ABB RobotStudio station: Cell5678 2025_5_GPA546_A0610_RW7.5.rspag

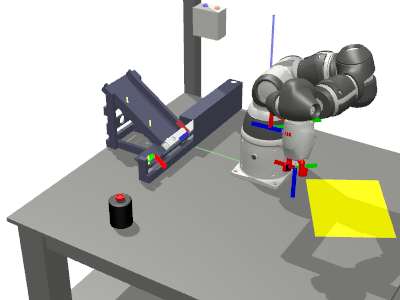
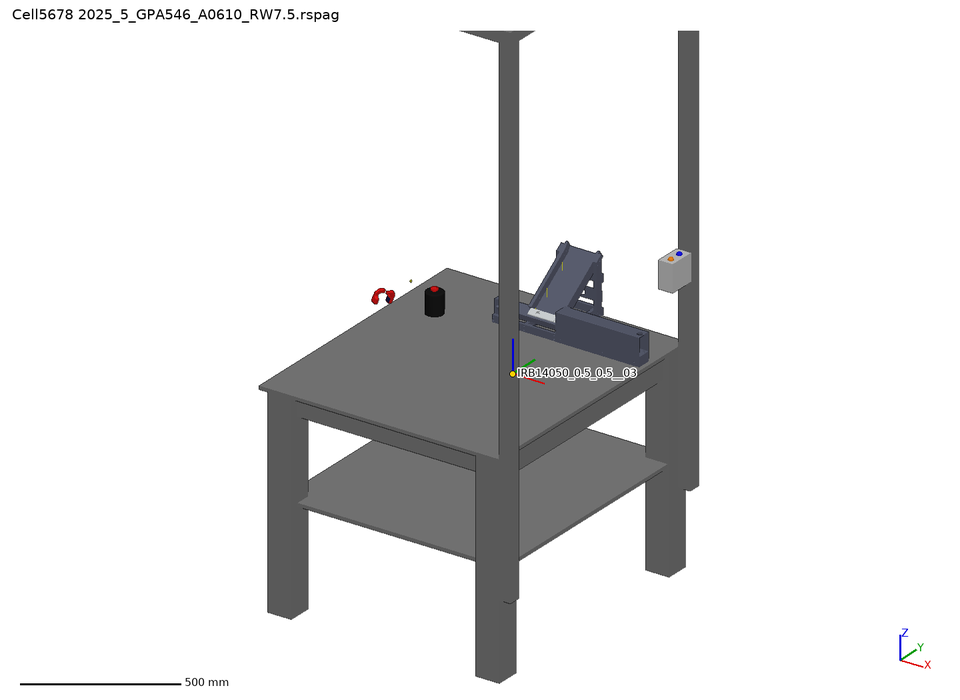
[picture v1: parts stored in the station drawn from their meshes, with robot base, taught points and paths (robot models come from the ABB library and are not in the file)]
--- station ---
Station Cell5678 011021_GPA546_A0610_publ5_1 (saved by RobotStudio 24.2.10821.1)
Controller IRB14050
  mechanical unit ROB_1: IRB14050_0.5_0.5__03, 6 joints, base frame (0, 0, 0) mm
  mechanical unit ROB_1_7: IRB14050_0.5_0.5__03, 1 joints, base frame (0, 0, 0) mm
Layout (positions relative to the parent item):
  - IRB14050_0.5_0.5__03 [mechanism, from %ABB.RobotStudio.Models.IRB14050%\IRB14050_0.5_0.5__03.rslib] at (0, 0, 0) mm; joint values [1.5708, -1.309, 1.5708, 0.3491, -1.5708, -1.2217, 1.5708] (rad or m)
  - Table 1020X900 [part] at (311.38, -523.15, 0.9) mm, rotated rx 0 ry 0 rz 90 deg, size 1020 x 954.9 x 2265 mm
  - Boite Lumière [part] at (359.1, 353.08, 238.5) mm, rotated rx 0 ry 0 rz 90 deg, size 100 x 55 x 100 mm
  - Glissoire_4 [part] at (-154.02, 493.45, 6.79) mm, rotated rx 0 ry 0 rz -90 deg, size 257.5 x 560.4 x 225.6 mm
  - Piston [mechanism, from Libraries\Piston.rslib] at (-154.02, 493.45, 6.79) mm, rotated rx 0 ry 0 rz -90 deg; joint values [0] (rad or m)
  - SC_Gestion_Lampes [smart component]
      signals: DI BlueLampOn, DI YellowLampOn
      connections:
        SC_Gestion_Lampes.BlueLampOn -> Highlighter.Active
        SC_Gestion_Lampes.YellowLampOn -> Highlighter_2.Active
    - Highlighter [smart component, from Components\Highlighter.rslib]
        properties: Object=Lumière Bleu; Color=[0 0 255]; Opacity=255
    - Highlighter_2 [smart component, from Components\Highlighter.rslib]
        properties: Object=Lumière Jaune; Color=[255 50 0]; Opacity=255
  - Lumière Bleu [part] at (10.6, -21.42, 0) mm, rotated rx 0 ry 0 rz -90 deg, size 19.9 x 19.9 x 20 mm
  - Lumière Jaune [part] at (10.6, -21.42, 0) mm, rotated rx 0 ry 0 rz -90 deg, size 19.9 x 19.9 x 20 mm
  - SC_Gestion poussoir [smart component] at (-154.05, 492.67, 6.82) mm, rotated rx 0 ry 0 rz -90 deg
      properties: PartAtPickPoint=(none)
      signals: DI ValveON, DO AtExtend, DO AtRetract, AO BlocAtLow, DO BlocAtHigh, DO NoHoleDetect, DO BlocZS0101, DI Orientation
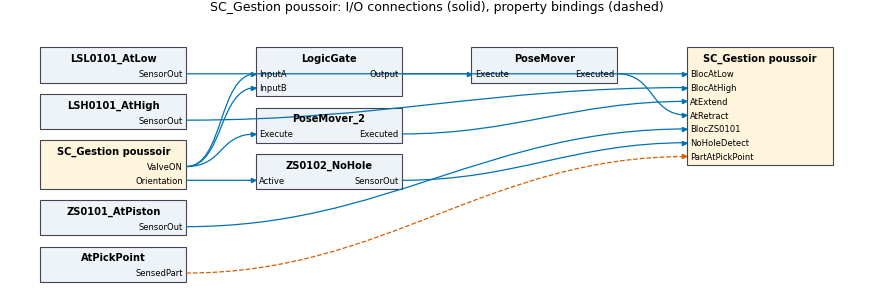
      connections:
        LSL0101_AtLow.SensorOut -> SC_Gestion poussoir.BlocAtLow
        LSH0101_AtHigh.SensorOut -> SC_Gestion poussoir.BlocAtHigh
        LogicGate.Output -> PoseMover.Execute
        SC_Gestion poussoir.ValveON -> LogicGate.InputA
        SC_Gestion poussoir.ValveON -> LogicGate.InputB
        SC_Gestion poussoir.ValveON -> PoseMover_2.Execute
        PoseMover_2.Executed -> SC_Gestion poussoir.AtExtend
        PoseMover.Executed -> SC_Gestion poussoir.AtRetract
        ZS0101_AtPiston.SensorOut -> SC_Gestion poussoir.BlocZS0101
        SC_Gestion poussoir.Orientation -> ZS0102_NoHole.Active
        ZS0102_NoHole.SensorOut -> SC_Gestion poussoir.NoHoleDetect
        AtPickPoint.SensedPart => SC_Gestion poussoir.PartAtPickPoint
    - PoseMover [smart component, from Components\PoseMover.rslib] at (516.34, -722.56, -751.2) mm, rotated rx 0 ry 0 rz -5.2 deg
        properties: Mechanism=Piston; Pose=2; Duration=2
    - PoseMover_2 [smart component, from Components\PoseMover.rslib] at (516.34, -722.56, -751.2) mm, rotated rx 0 ry 0 rz -5.2 deg
        properties: Mechanism=Piston; Pose=3; Duration=2
    - LogicGate [smart component, from Components\LogicGate.rslib] at (516.34, -722.56, -751.2) mm, rotated rx 0 ry 0 rz -5.2 deg
        properties: Operator=NOT; Delay=0
    - ZS0101_AtPiston [smart component, from Components\LineSensor.rslib] at (516.34, -722.56, -751.2) mm, rotated rx 0 ry 0 rz -5.2 deg
        properties: Start=[-0.375541 0.733962 0.796662]; End=[-0.375541 0.733962 0.826662]; Radius=0.001; SensedPart=Bloc_ETS_D0; SensedPoint=[-0.111608673095703 0.283746734619141 0.0522771530151367]; Length=0.03; Tag=(none)
      - _sensorPart_ [part], size 2 x 2 x 30 mm
    - LSL0101_AtLow [smart component, from Components\LineSensor.rslib] at (516.34, -722.56, -751.2) mm, rotated rx 0 ry 0 rz -5.2 deg
        properties: Start=[-0.437628 0.727535 0.840369]; End=[-0.437628 0.727535 0.870369]; Radius=0.001; SensedPart=(none); SensedPoint=[0 0 0]; Length=0.0299999999999999; Tag=(none)
      - _sensorPart_ [part], size 2 x 2 x 30 mm
    - LSH0101_AtHigh [smart component, from Components\LineSensor.rslib] at (516.34, -722.56, -751.2) mm, rotated rx 0 ry 0 rz -5.2 deg
        properties: Start=[-0.520412 0.718966 0.898644]; End=[-0.520412 0.718966 0.928644]; Radius=0.001; SensedPart=(none); SensedPoint=[0 0 0]; Length=0.03; Tag=(none)
      - _sensorPart_ [part], size 2 x 2 x 30 mm
    - ZS0102_NoHole [smart component, from Components\LineSensor.rslib] at (516.34, -722.56, -751.2) mm, rotated rx 0 ry 0 rz -5.2 deg
        properties: Start=[-0.38024951999447 0.783345123820164 0.800380266534001]; End=[-0.367482382887285 0.784507947657669 0.818689278845135]; Radius=0.004; SensedPart=Bloc_ETS_G0; SensedPoint=[-0.0620019989013672 0.283955902099609 0.0559951324462891]; Length=0.0223511046930568; Tag=(none)
      - _sensorPart_ [part], size 19.3 x 9.1 x 22.9 mm
    - AtPickPoint [smart component, from Components\LineSensor.rslib] at (516.34, -722.56, -751.2) mm, rotated rx 0 ry 0 rz -5.2 deg
        properties: Start=[-0.358924 0.623964 0.79302]; End=[-0.358924 0.623964 0.82302]; Radius=0.001; SensedPart=(none); SensedPoint=[0 0 0]; Length=0.03; Tag=(none)
      - _sensorPart_ [part], size 2 x 2 x 30 mm
  - SC_Gestion bloc [smart component]
      signals: DI PistonValve_ON, DI PistonRetracted, DO SimulBlocPoussoir, DI PistonExtended, DI Reinit_Droite, DI Reinit_Gauche, DI Initialisation
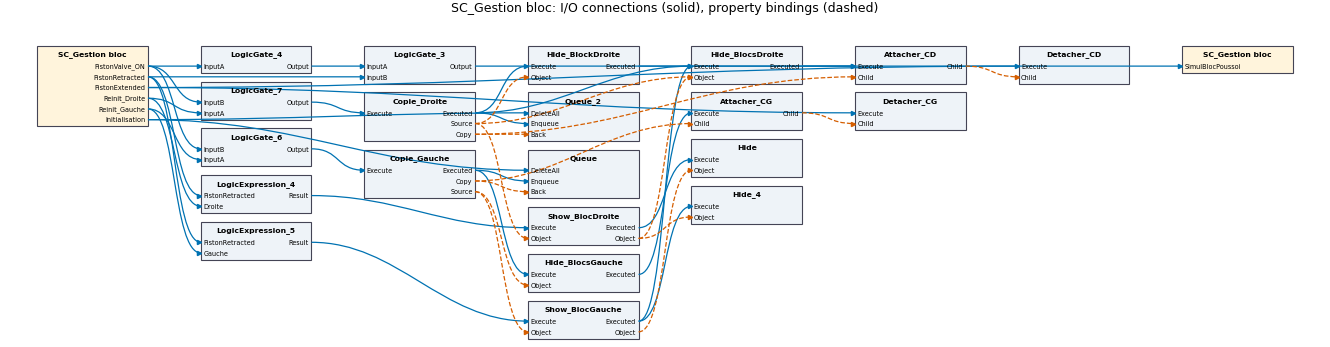
      connections:
        SC_Gestion bloc.PistonValve_ON -> LogicGate_4.InputA
        LogicGate_3.Output -> SC_Gestion bloc.SimulBlocPoussoir
        LogicExpression_4.Result -> Show_BlocDroite.Execute
        LogicExpression_5.Result -> Show_BlocGauche.Execute
        SC_Gestion bloc.PistonRetracted -> LogicExpression_4.PistonRetracted
        SC_Gestion bloc.PistonRetracted -> LogicExpression_5.PistonRetracted
        Copie_Gauche.Executed -> Hide_BlocsGauche.Execute
        SC_Gestion bloc.PistonExtended -> Detacher_CG.Execute
        LogicGate_6.Output -> Copie_Gauche.Execute
        SC_Gestion bloc.PistonValve_ON -> LogicGate_6.InputB
        LogicGate_7.Output -> Copie_Droite.Execute
        SC_Gestion bloc.PistonValve_ON -> LogicGate_7.InputB
        SC_Gestion bloc.PistonExtended -> Detacher_CD.Execute
        SC_Gestion bloc.Reinit_Droite -> LogicExpression_4.Droite
        SC_Gestion bloc.Reinit_Gauche -> LogicExpression_5.Gauche
        LogicGate_4.Output -> LogicGate_3.InputA
        SC_Gestion bloc.PistonRetracted -> LogicGate_3.InputB
        SC_Gestion bloc.Reinit_Gauche -> LogicGate_6.InputA
        SC_Gestion bloc.Reinit_Droite -> LogicGate_7.InputA
        Copie_Droite.Executed -> Hide_BlocsDroite.Execute
        Hide_BlocsDroite.Executed -> Attacher_CD.Execute
        SC_Gestion bloc.Initialisation -> Queue.DeleteAll
        SC_Gestion bloc.Initialisation -> Queue_2.DeleteAll
        Show_BlocDroite.Executed -> Hide.Execute
        Show_BlocGauche.Executed -> Hide_2.Execute
        Hide_BlocsGauche.Executed -> Attacher_CG.Execute
        Copie_Droite.Executed -> Hide_BlockDroite.Execute
        Hide_BlockDroite.Executed -> Attacher_CD.Execute
        Show_BlocGauche.Executed -> Hide_4.Execute
        Copie_Gauche.Executed -> Queue.Enqueue
        Copie_Droite.Executed -> Queue_2.Enqueue
        Attacher_CG.Child => Detacher_CG.Child
        Attacher_CD.Child => Detacher_CD.Child
        Show_BlocGauche.Object => Hide.Object
        Show_BlocDroite.Object => Hide_2.Object
        Copie_Gauche.Copy => Attacher_CG.Child
        Copie_Gauche.Source => Hide_BlocsGauche.Object
        Copie_Gauche.Source => Show_BlocGauche.Object
        Copie_Droite.Source => Show_BlocDroite.Object
        Copie_Droite.Copy => Attacher_CD.Child
        Copie_Droite.Source => Hide_BlocsDroite.Object
        Copie_Droite.Source => Hide_BlockDroite.Object
        Show_BlocDroite.Object => Hide_4.Object
        Copie_Gauche.Copy => Queue.Back
        Copie_Droite.Copy => Queue_2.Back
    - LogicGate_3 [smart component, from Components\LogicGate.rslib]
        properties: Operator=AND; Delay=0
    - LogicGate_4 [smart component, from Components\LogicGate.rslib]
        properties: Operator=NOT; Delay=0
    - Show_BlocDroite [smart component, from Components\Show.rslib]
        properties: Object=Bloc_ETS_D0
    - Show_BlocGauche [smart component, from Components\Show.rslib]
        properties: Object=Bloc_ETS_G0
    - Hide_BlocsGauche [smart component, from Components\Hide.rslib]
        properties: Object=Bloc_ETS_G0
    - LogicExpression_4 [smart component, from Components\LogicExpression.rslib]
        properties: Expression=PistonRetracted and Droite
    - LogicExpression_5 [smart component, from Components\LogicExpression.rslib]
        properties: Expression=PistonRetracted and Gauche
    - Copie_Droite [smart component, from Components\Source.rslib]
        properties: Source=Bloc_ETS_D0; Copy=(none); Parent=(none); Position=[-0.079147 0.2595 0.06725]; Orientation=[0.610865238198015 0 0]; Transient=true; PhysicsBehavior=0
    - Copie_Gauche [smart component, from Components\Source.rslib]
        properties: Source=Bloc_ETS_G0; Copy=(none); Parent=(none); Position=[-0.079147 0.26106 0.06725]; Orientation=[-2.18166156499291 0 3.14159265358979]; Transient=true; PhysicsBehavior=0
    - Attacher_CG [smart component, from Components\Attacher.rslib]
        properties: Parent=L2; Flange=0; Child=(none); Mount=false; Offset=[0 0 0]; Orientation=[0 0 0]
    - Detacher_CG [smart component, from Components\Detacher.rslib]
        properties: Child=(none); KeepPosition=true
    - LogicGate_6 [smart component, from Components\LogicGate.rslib]
        properties: Operator=AND; Delay=0
    - LogicGate_7 [smart component, from Components\LogicGate.rslib]
        properties: Operator=AND; Delay=0
    - Attacher_CD [smart component, from Components\Attacher.rslib]
        properties: Parent=L2; Flange=0; Child=(none); Mount=false; Offset=[0 0 0]; Orientation=[0 0 0]
    - Detacher_CD [smart component, from Components\Detacher.rslib]
        properties: Child=(none); KeepPosition=true
    - Queue [smart component, from Components\Queue.rslib]
        properties: Back=(none); Front=(none); Queue=; NumberOfObjects=0
    - Queue_2 [smart component, from Components\Queue.rslib]
        properties: Back=(none); Front=(none); Queue=; NumberOfObjects=0
    - Hide [smart component, from Components\Hide.rslib]
        properties: Object=Bloc_ETS_G0
    - Hide_BlockDroite [smart component, from Components\Hide.rslib]
        properties: Object=Bloc_ETS_D0
    - Hide_4 [smart component, from Components\Hide.rslib]
        properties: Object=Bloc_ETS_D0
  - Feuille8.5x11 [part, from Libraries\Feuille8.5x11.rslib] at (-117.65, -454.21, 2) mm, rotated rx 0 ry 0 rz 30 deg
  - Smart_Gripper_Group [graphiccomponentgroup] at (-291.1, -222.85, 372.1) mm, rotated rx -165.24 ry 14.08 rz 69.35 deg
    - YuMiFinger_2 [part] at (-0.5, -6.5, 84) mm, rotated rx 0 ry 0 rz 180 deg, size 33.9 x 23.8 x 46.2 mm
    - Smart_Gripper [mechanism] at (0, 0, 0) mm; joint values [0.025] (rad or m)
        TCP Servo at (0, 0, 84) mm
        TCP VaccumOne at (63.5, 18.5, 37.5) mm, rotated rx 0 ry 90 rz 0 deg
        TCP Camera at (-7.3, 28.3, 35.1) mm, rotated rx 0 ry 90 rz 90 deg
        links: HandBase, DownFinger, UpFinger
    - YuMiFinger [part] at (0.5, 6.5, 84) mm, size 33.9 x 23.8 x 46.2 mm
  - CrayonAttache [part] at (-176.86, -64.88, 338.21) mm, rotated rx -31.34 ry -80.07 rz -136.95 deg, size 25 x 25 x 53.7 mm
  - Support_Probe [part] at (-446.5, 212.7, 77.11) mm, size 63.4 x 63.5 x 76.2 mm
  - CrayonDansSupport [part] at (-446.94, 212.7, 84.94) mm, rotated rx 180 ry 0 rz 180 deg, size 25 x 25 x 53.7 mm
  - PadUp [part] at (-346.78, -144.15, -46.95) mm, rotated rx 5.22 ry 23.93 rz 58.66 deg, size 8.7 x 19.9 x 17.8 mm
  - PadDown [part] at (-330.6, -100.22, -58.38) mm, rotated rx 5.22 ry 23.93 rz 58.66 deg, size 8.7 x 19.9 x 17.8 mm
  - Bloc_ETS_G0 [part] at (-79.15, 261.06, 67.25) mm, rotated rx -125 ry 0 rz 180 deg, size 99.6 x 26.5 x 26.5 mm
  - SC_Gestion crayon [smart component]
      signals: DI Succion
      connections:
        ObjectComparer.Output -> LogicGate.InputB
        SC_Gestion crayon.Succion -> LogicGate.InputA
        LogicGate.Output -> Attacher.Execute
        SC_Gestion crayon.Succion -> LogicGate_2.InputA
        LogicGate_2.Output -> Detacher.Execute
        LineSensor.SensedPart => ObjectComparer.ObjectB
        DetecteurCrayon.SensedPart => ObjectComparer_2.ObjectB
        DetecteurCrayon.SensedPart => ObjectComparer_3.ObjectB
        DetecteurCrayon.SensedPart => GetParent.Child
        DetecteurCrayon.SensedPart => ObjectComparer.ObjectB
        ObjectComparer.ObjectA => Attacher.Child
        ObjectComparer.ObjectA => Detacher.Child
    - DetecteurCrayon [smart component, from Components\VolumeSensor.rslib] at (-291.1, -222.85, 372.1) mm, rotated rx -165.24 ry 14.08 rz 69.35 deg
        properties: CornerPoint=[0.0651107378011944 0.0208370386716533 0.0417702285630413]; Orientation=[-1.57722951002103 0.179635421049669 -1.58129130311226]; Length=0.008; Width=0.008; Height=0.001; PartialHit=true; SensedPart=Pneumatic; Tag=(none)
      - _sensorPart_ [part], size 1.1 x 9.3 x 9.3 mm
    - ObjectComparer [smart component, from Components\ObjectComparer.rslib]
        properties: ObjectA=CrayonDansSupport; ObjectB=Pneumatic
    - LogicGate [smart component, from Components\LogicGate.rslib]
        properties: Operator=AND; Delay=0
    - Attacher [smart component, from Components\Attacher.rslib]
        properties: Parent=Pneumatic; Flange=0; Child=CrayonDansSupport; Mount=false; Offset=[0 0 0]; Orientation=[0 0 0]
    - LogicGate_2 [smart component, from Components\LogicGate.rslib]
        properties: Operator=NOT; Delay=0
    - Detacher [smart component, from Components\Detacher.rslib]
        properties: Child=CrayonDansSupport; KeepPosition=true
  - LogicGate [smart component, from Components\LogicGate.rslib]
      properties: Operator=OR; Delay=0
  - Random [smart component, from Components\Random.rslib]
      properties: Value=0.33026239151613; Min=0; Max=1
  - LogicGate_2 [smart component, from Components\LogicGate.rslib]
      properties: Operator=NOT; Delay=0
  - Bloc_ETS_D0 [part] at (-79.15, 281.54, 81.59) mm, rotated rx -55 ry 0 rz 0 deg, size 98 x 25.4 x 25.4 mm
  - ExecuteCommand [smart component, from Components\ExecuteCommand.rslib]
      properties: CommandID=ProgramSetPPMain
Attachment: YuMiFinger_2 is attached to Smart_Gripper / UpFinger
Attachment: YuMiFinger is attached to Smart_Gripper / DownFinger
Attachment: Smart_Gripper_Group is attached to IRB14050_0.5_0.5__03 / Link7
Attachment: PadUp is attached to YuMiFinger_2
Attachment: DetecteurCrayon is attached to Pneumatic
Attachment: Bloc_ETS_G0 is attached to Piston / L2
Attachment: Bloc_ETS_D0 is attached to Piston / L2
Attachment: PadDown is attached to YuMiFinger
EventTableEntry 1381: Group=, Trigger=CabinetIO_0_DO9_FV0101 1382, Actions=[EventTableActionMechanicalPose 1383, st_PistonIn 1393], Comment=, ActivationMode=2, Cyclic=false
EventTableTriggerIO 1382: IOValue=[1], IRC5Controller=? -1, Operator=0, SignalSource=IRB14050 515
EventTableActionMechanicalPose 1383: VirtualSignal=st_PistonOut, Mechanism=Piston 1047, ToPoseName=OUT, VirtualSignalValue=[1]
EventTableEntry 1384: Group=, Trigger=st_PistonOut 1385, Actions=[CabinetIO_0_DI14_ZS0104 1386], Comment=, ActivationMode=2, Cyclic=false
EventTableTriggerIO 1385: IOValue=[1], IRC5Controller=? -1, Operator=0, SignalSource=Cell5678 011021_GPA546_A0610_publ5_1 1
EventTableActionIO 1386: IOValue=[1], IRC5Controller=? -1, SignalTarget=IRB14050 515
EventTableEntry 1387: Group=, Trigger=CabinetIO_0_DO9_FV0101 1388, Actions=[EventTableActionMechanicalPose 1389, st_PistonOut 1394], Comment=, ActivationMode=2, Cyclic=false
EventTableTriggerIO 1388: IOValue=[0], IRC5Controller=? -1, Operator=0, SignalSource=IRB14050 515
EventTableActionMechanicalPose 1389: VirtualSignal=st_PistonIn, Mechanism=Piston 1047, ToPoseName=IN, VirtualSignalValue=[1]
EventTableEntry 1390: Group=, Trigger=st_PistonIn 1391, Actions=[CabinetIO_0_DI13_ZS0103 1392], Comment=, ActivationMode=2, Cyclic=false
EventTableTriggerIO 1391: IOValue=[1], IRC5Controller=? -1, Operator=0, SignalSource=Cell5678 011021_GPA546_A0610_publ5_1 1
EventTableActionIO 1392: IOValue=[1], IRC5Controller=? -1, SignalTarget=IRB14050 515
EventTableActionIO 1393: IOValue=[0], IRC5Controller=? -1, SignalTarget=Cell5678 011021_GPA546_A0610_publ5_1 1
EventTableActionIO 1394: IOValue=[0], IRC5Controller=? -1, SignalTarget=Cell5678 011021_GPA546_A0610_publ5_1 1
EventTableEntry 1403: Group=, Trigger=custom_DO_0_gClose 1404, Actions=[EventTableActionMechanicalPose 1405, st_Detach 1415], Comment=, ActivationMode=2, Cyclic=false
EventTableTriggerIO 1404: IOValue=[1], IRC5Controller=? -1, Operator=0, SignalSource=IRB14050 515
EventTableActionMechanicalPose 1405: VirtualSignal=st_Attach, Mechanism=Smart_Gripper 1837, ToPoseName=FermeBloc, VirtualSignalValue=[1]
EventTableEntry 1406: Group=, Trigger=custom_DO_1_gOpen 1407, Actions=[EventTableActionMechanicalPose 1408, st_Attach 1416], Comment=, ActivationMode=2, Cyclic=false
EventTableTriggerIO 1407: IOValue=[1], IRC5Controller=? -1, Operator=0, SignalSource=IRB14050 515
EventTableActionMechanicalPose 1408: VirtualSignal=st_Detach, Mechanism=Smart_Gripper 1837, ToPoseName=SyncPosition, VirtualSignalValue=[1]
EventTableEntry 1409: Group=, Trigger=st_Attach 1410, Actions=[EventTableActionAttach 1411], Comment=, ActivationMode=2, Cyclic=false
EventTableTriggerIO 1410: IOValue=[1], IRC5Controller=? -1, Operator=0, SignalSource=Cell5678 011021_GPA546_A0610_publ5_1 1
EventTableActionAttach 1411: AttachmentParent=Smart_Gripper 1837, AttachmentChild=? -1, MountObject=false, Offset=[X=1, Y=0, Z=0, W=0, X=0, Y=1, Z=0, W=0, X=0, Y=0, Z=1, W=0, X=0, Y=0, Z=0, W=1], FlangeIndext=0, FindNearest=true
EventTableEntry 1412: Group=, Trigger=st_Detach 1413, Actions=[EventTableActionDetach 2269], Comment=, ActivationMode=2, Cyclic=false
EventTableTriggerIO 1413: IOValue=[1], IRC5Controller=? -1, Operator=0, SignalSource=Cell5678 011021_GPA546_A0610_publ5_1 1
EventTableActionIO 1415: IOValue=[0], IRC5Controller=? -1, SignalTarget=Cell5678 011021_GPA546_A0610_publ5_1 1
EventTableActionIO 1416: IOValue=[0], IRC5Controller=? -1, SignalTarget=Cell5678 011021_GPA546_A0610_publ5_1 1
EventTableActionDetach 2269: AttachmentParent=Smart_Gripper 1837, AttachmentChild=? -1
Station signals: DI st_PistonOut, DI st_PistonIn, DI st_Attach, DI st_Detach, DO SimulBlocPoussoir, DI Initialisation
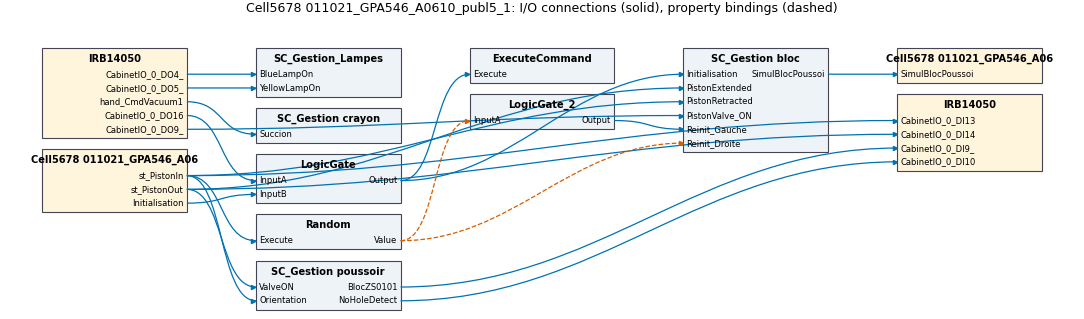
Station logic (signal -> signal, property => property):
  IRB14050.CabinetIO_0_DO4_JB01_LampBlu -> SC_Gestion_Lampes.BlueLampOn
  IRB14050.CabinetIO_0_DO5_JB01_LampOr -> SC_Gestion_Lampes.YellowLampOn
  Cell5678 011021_GPA546_A0610_publ5_1.st_PistonIn -> IRB14050.CabinetIO_0_DI13_ZS0103
  Cell5678 011021_GPA546_A0610_publ5_1.st_PistonOut -> IRB14050.CabinetIO_0_DI14_ZS0104
  IRB14050.hand_CmdVacuum1 -> SC_Gestion crayon.Succion
  SC_Gestion bloc.SimulBlocPoussoir -> Cell5678 011021_GPA546_A0610_publ5_1.SimulBlocPoussoir
  IRB14050.CabinetIO_0_DO16 -> LogicGate.InputA
  LogicGate.Output -> SC_Gestion bloc.Initialisation
  Cell5678 011021_GPA546_A0610_publ5_1.st_PistonOut -> SC_Gestion bloc.PistonExtended
  SC_Gestion poussoir.BlocZS0101 -> IRB14050.CabinetIO_0_DI9_ZS0101
  Cell5678 011021_GPA546_A0610_publ5_1.st_PistonOut -> SC_Gestion poussoir.ValveON
  Cell5678 011021_GPA546_A0610_publ5_1.st_PistonIn -> SC_Gestion bloc.PistonRetracted
  IRB14050.CabinetIO_0_DO9_FV0101 -> SC_Gestion bloc.PistonValve_ON
  Cell5678 011021_GPA546_A0610_publ5_1.st_PistonIn -> Random.Execute
  LogicGate_2.Output -> SC_Gestion bloc.Reinit_Gauche
  SC_Gestion poussoir.NoHoleDetect -> IRB14050.CabinetIO_0_DI10_ZS0102
  Cell5678 011021_GPA546_A0610_publ5_1.st_PistonIn -> SC_Gestion poussoir.Orientation
  Cell5678 011021_GPA546_A0610_publ5_1.Initialisation -> LogicGate.InputB
  LogicGate.Output -> ExecuteCommand.Execute
  Random.Value => SC_Gestion bloc.Reinit_Droite
  Random.Value => LogicGate_2.InputA
Targets, tools, work objects and paths stored in the station and not in the controller backup, written as RAPID:
! task T_ROB1
MODULE user
  PERS tooldata tPince:=[TRUE,[[0,0,114.2],[1,0,0,0]],[0.229,[7.9,12.4,48.7],[1,0,0,0],0.00021,0.00023,0.00008]];
  PERS tooldata tVentouse:=[TRUE,[[63.5,18.5,37.5],[0.707107,0,0.707107,0]],[0.24,[8.2,12.5,48.1],[1,0,0,0],0.00022,0.00024,0.00009]];
  PERS tooldata tCrayon:=[TRUE,[[118.5,18.5,37.5],[0.707107,0,0.707107,0]],[0.24,[8.2,12.5,48.1],[1,0,0,0],0.00022,0.00024,0.00009]];
ENDMODULE


--- Backups/IRB14050/RAPID/TASK1/PROGMOD/Demo.modx ---
MODULE Demo

!@@@@@@@@@@@@@@@@@@@ IMPORTANT @@@@@@@@@@@@@@@@@
! Pour ouvrir la pince sur le simulateur: Pince_Ouvre;
! Pour fermer la pince sur le simulateur: Pince_Ferme;
! Pour ouvrir la pince sur le vrai robot Yumi: g_GripOut;
! Pour fermer la pince sur le vrai robot Yumi: g_GripIn;
!@@@@@@@@@@@@@@@@@@@@@@@@@@@@@@@@@@@@@@@@@@@@@@@

! -------------------------------------------------------------------------------------
! Programme : Demo
! Auteurs : _______________ ET ______________
! Date : _________________
! Révision : ________________
!
! Description :
! Ce programme permet de prendre deux blocs dans une glissoire et de les
! superposer sur une table de travail, avec les trous dans le même sens.
! -------------------------------------------------------------------------------------


  ! "Positions" à peufiner sur le vrai robot
  PERS robtarget rCrayon:=[[-446.844,212.768,88],[0,0.92388,-0.382683,0],[0,0,0,5],[13.6937,9E+9,9E+9,9E+9,9E+9,9E+9]];
  PERS robtarget rGlissoire:=[[-193.434,277.819,65.0723],[0.212106,-0.671728,0.677924,0.210267],[0,0,2,5],[-88.7724,9E+9,9E+9,9E+9,9E+9,9E+9]];
  PERS jointtarget jRetrait:=[[90,-75,20,-90,-70,90],[90,9E+09,9E+09,9E+09,9E+09,9E+09]];
  PERS robtarget rDepot:= [[-285.818,-59.2446,23.85],[0,-0.707107,0.707107,0],[0,1,0,5],[-63.0892,9E+9,9E+9,9E+9,9E+9,9E+9]];

  ! Donnees de type "positions" calculées
  VAR robtarget rDepot2;

  ! Donnees de type constante
  CONST num Epaisseur:=1; ! Épaisseur d'un bloc (en pouces)
  CONST num PouceToMM:=25.4; ! Facteur de conversion
  CONST num Decalage:=200; ! Distance d'approche ou de retrait (mm)

  ! Données de type variable
  VAR num EpaisMM:=0;


  ! Vitesse d'approche et de retrait (mm/sec)
  CONST speeddata LowSpeed:=[250,500,5000,1000];

  ! Vitesse maximale du robot (mm/sec)
  CONST speeddata HighSpeed:=[1000,500,5000,1000];

  ! Etat des entrees/sorties
  CONST dionum Ouverte:=0;
  CONST dionum Fermee:=1;
  CONST dionum Retracte:=0;
  CONST dionum Extension:=1;

! -------------------------------------------------------------------------------------
! Procedure : main
! -------------------------------------------------------------------------------------
PROC main()

	! 1) Initialisation :
	init;

	! Deplacement à retrait
	MoveAbsJ jRetrait, HighSpeed, fine, tPince\wobj:=wobj0;

	! 2) Calculs :
	EpaisMM := Epaisseur * PouceToMM; ! Conversion en mm
	rDepot2 := Offs(rDepot,0,0,EpaisMM);

	! 3) Déplacement du premier bloc :
	! Prise du bloc dans le glissoire
	Prise;
	! Dépôt du bloc 1 à la localisation rDepot :
	Depot(rDepot);

	! 4) Déplacement du deuxième bloc :
	! Prise du bloc dans le glissoire
    Prise;
	! Dépôt du bloc 2 à la localisation rDepot :
	Depot(rDepot2);

	! 5) Retourner à retrait
	MoveAbsJ jRetrait,HighSpeed,z50,tPince\wobj:=wobj0;

	Pince_Ouvre;
    SetDO CabinetIO_0_DO16,1; ! ramasse-les-blocs dans la simulation
    WaitTime 2;
    SetDO CabinetIO_0_DO16,0; ! ramasse-les-blocs dans la simulation

ENDPROC

! -------------------------------------------------------------------------------------
! Procedure : init
! -------------------------------------------------------------------------------------
PROC init()

    ! Initialisation du Smart gripper
    !g_Calibrate \Jog;
    G_init \Calibrate;

	VelSet 25,1000; ! Limitation imposée pour la sécurité, obligatoire

	SetDO CabinetIO_0_DO9_FV0101, Retracte; ! Rentrer le vérin

    ! Ouvrir la pince
    Pince_Ouvre;
    WaitTime 2;

ENDPROC

! -------------------------------------------------------------------------------------
! Procédure : Prise
! Description : S'approcher de la glissoire, attendre une pièce dans la glissoire,
! l'indexer, la prendre de manière sécuritaire
! -------------------------------------------------------------------------------------
PROC Prise()

    VAR robtarget rGlissoireCalc;

    ! Vérification de la présence d'un bloc dans la glissoire
	IF CabinetIO_0_DI9_ZS0101 = 0 THEN
		TPErase;
		TPWrite "Aucun bloc dans la glissoire";
		TPWrite "Placer deux blocs et remettre en mode AUTO";
		WaitDI CabinetIO_0_DI9_ZS0101, 1; ! Attente d'un bloc
		Waittime 1; ! attente que le bloc se stabilise
	ENDIF

    ! Prendre le bloc de la même façon par rapport au trou
    IF CabinetIO_0_DI10_ZS0102 = 1 THEN
    	rGlissoireCalc := RelTool(rGlissoire, 0, 0, 0 \Rz := 180);
        rGlissoireCalc.robconf.cf6 := 0;
    ELSE
    	rGlissoireCalc := rGlissoire;
    ENDIF

    ! Préhension du bloc
    ConfJ \Off;
    ConfL \Off;
    MoveAbsJ jRetrait, HighSpeed, z50,tPince\wobj:=wobj0;
	MoveJ RelTool(rGlissoireCalc,0,0,-Decalage),HighSpeed,z50,tPince\wobj:=wobj0;
	SetDO CabinetIO_0_DO9_FV0101, Extension; ! Pousser le bloc
	WAITDI CabinetIO_0_DI14_ZS0104,1; ! Attendre que le vérin soit complètement sorti
	MoveL rGlissoireCalc, LowSpeed, fine, tPince\wobj:=wobj0;

	SetDO CabinetIO_0_DO9_FV0101, Retracte;
    !WAITDI CabinetIO_0_DI14_ZS0104,0;
	 WAITDI CabinetIO_0_DI13_ZS0103,1;
    !g_GripIn; ! Fermer la pince
    Pince_Ferme;

	MoveL RelTool(rGlissoireCalc,0,0,-Decalage),LowSpeed,z50,tPince\wobj:=wobj0;

ENDPROC

! -------------------------------------------------------------------------------------
! Procédure : Depot
! Argument : Reçoit un robtarget indiquant où placer un bloc, avec une approche et
! un dégagement.
! -------------------------------------------------------------------------------------
PROC Depot(robtarget rPosDepot)

    ! Même si rPosDepot a élé enseigné, en mettant les conf à Off, le robot fait
    ! moins de mouvements inutiles
    ConfJ \Off;
	MoveJ RelTool(rPosDepot,0,0,-Decalage), HighSpeed, z50, tPince\wobj:=wobj0;
    ConfL \Off;
	MoveL rPosDepot, LowSpeed, fine, tPince;

    !g_GripOut;! Ouvrir la pince
    !g_stop;
    Pince_Ouvre;
	MoveL RelTool(rPosDepot,0,0,-Decalage), LowSpeed, z50, tPince\wobj:=wobj0;

ENDPROC

! -------------------------------------------------------------------------------------
! Utilisez ces deux procédures pour fermer ou ouvrir la pince de Yumi.
! Sur le vrai robot, utilisez les commandes g_GripIn et g_GripOut
! -------------------------------------------------------------------------------------
PROC Pince_Ferme()
    SetDO custom_DO_0_gClose,1;
    SetDO custom_DO_1_gOpen,0;
    !g_GripIn;
    WaitTime 1.5;
ENDPROC

PROC Pince_Ouvre()
     SetDO custom_DO_1_gOpen,1;
     SetDO custom_DO_0_gClose,0;
     !g_GripOut;
     WaitTime 1.5;
ENDPROC


ENDMODULE

--- Backups/IRB14050/SYSPAR/EIO.cfg ---
EIO:CFG_1.0:7:0::
#
EIO_CROSS:

      -Name "Cross_Signal_Lamp" -Res "Signal_Lamp" -Act1 "scDriveEnable"
#
EIO_SIGNAL_SAFELEVEL:

      -Name "FlangePowerSafeLevel" -ActionWhenStartup "Last"

      -Name "SGcmdSafeLevel" -ActionWhenAccessible "Default"
#
ETHERNETIP_DEVICE:

      -Name "ManipulatorIO" -VendorName "ABB Robotics" -ProductName "DSQC1030"\
      -Label "ABB Manipulator I/O Device" -Address "192.168.125.101"\
      -VendorId 75 -ProductCode 29 -DeviceType 12 -OutputAssembly 100\
      -InputAssembly 101 -ConfigurationAssembly 102\
      -ConnectionPriority "SCHEDULE" -OutputSize 2 -InputSize 2\
      -ConfigurationSize 8\
      -ConfigurationData00 "01 02 09 10 01 08 10 01 00 00 00 00 00 00 00 00"\
      -O2T_RPI 40000 -T2O_RPI 40000

      -Name "Hand" -VendorName "ABB" -ProductName "EtherNet/IP EIP" -Label "2"\
      -Address "192.168.125.30" -VendorId 75 -ProductCode 1 -OutputAssembly 100\
      -InputAssembly 101 -OutputSize 10 -InputSize 10 -O2T_RPI 10000\
      -T2O_RPI 10000 -ConnectionTimeoutMultiplier 2

      -Name "CabinetIO" -VendorName "ABB Robotics" -ProductName "DSQC1030"\
      -Label "ABB Local I/O Device" -Address "192.168.125.100" -VendorId 75\
      -ProductCode 29 -DeviceType 12 -OutputAssembly 100 -InputAssembly 101\
      -ConfigurationAssembly 102 -ConnectionPriority "SCHEDULE" -OutputSize 2\
      -InputSize 2 -ConfigurationSize 8\
      -ConfigurationData00 "01 02 09 10 01 08 10 01 00 00 00 00 00 00 00 00"\
      -O2T_RPI 40000 -T2O_RPI 40000
#
EIO_SIGNAL:

      -Name "custom_DI_0" -SignalType "DI" -Device "ManipulatorIO"\
      -DeviceMap "8" -Access "All"

      -Name "custom_DI_1" -SignalType "DI" -Device "ManipulatorIO"\
      -DeviceMap "9" -Access "All"

      -Name "custom_DI_2" -SignalType "DI" -Device "ManipulatorIO"\
      -DeviceMap "10" -Access "All"

      -Name "custom_DI_3" -SignalType "DI" -Device "ManipulatorIO"\
      -DeviceMap "11" -Access "All"

      -Name "custom_DI_4" -SignalType "DI" -Device "ManipulatorIO"\
      -DeviceMap "12" -Access "All"

      -Name "custom_DI_5" -SignalType "DI" -Device "ManipulatorIO"\
      -DeviceMap "13" -Access "All"

      -Name "custom_DI_6" -SignalType "DI" -Device "ManipulatorIO"\
      -DeviceMap "14" -Access "All"

      -Name "custom_DI_7" -SignalType "DI" -Device "ManipulatorIO"\
      -DeviceMap "15" -Access "All"

      -Name "custom_DO_0_gClose" -SignalType "DO" -Device "ManipulatorIO"\
      -DeviceMap "8" -Access "All"

      -Name "custom_DO_1_gOpen" -SignalType "DO" -Device "ManipulatorIO"\
      -DeviceMap "9" -Access "All"

      -Name "custom_DO_2" -SignalType "DO" -Device "ManipulatorIO"\
      -DeviceMap "10" -Access "All"

      -Name "custom_DO_3" -SignalType "DO" -Device "ManipulatorIO"\
      -DeviceMap "11" -Access "All"

      -Name "custom_DO_4" -SignalType "DO" -Device "ManipulatorIO"\
      -DeviceMap "12" -Access "All"

      -Name "custom_DO_5" -SignalType "DO" -Device "ManipulatorIO"\
      -DeviceMap "13" -Access "All"

      -Name "custom_DO_6" -SignalType "DO" -Device "ManipulatorIO"\
      -DeviceMap "14" -Access "All"

      -Name "custom_DO_7" -SignalType "DO" -Device "ManipulatorIO"\
      -DeviceMap "15" -Access "All"

      -Name "flange_24V" -SignalType "DO" -Device "ManipulatorIO" -DeviceMap "0"\
      -SafeLevel "FlangePowerSafeLevel"

      -Name "Signal_Lamp" -SignalType "DO" -Device "ManipulatorIO"\
      -DeviceMap "7"

      -Name "hall_sensor_joint_1" -SignalType "DI" -Device "ManipulatorIO"\
      -DeviceMap "0"

      -Name "hall_sensor_joint_2" -SignalType "DI" -Device "ManipulatorIO"\
      -DeviceMap "1"

      -Name "hall_sensor_joint_3" -SignalType "DI" -Device "ManipulatorIO"\
      -DeviceMap "3"

      -Name "hall_sensor_joint_4" -SignalType "DI" -Device "ManipulatorIO"\
      -DeviceMap "4"

      -Name "hall_sensor_joint_5" -SignalType "DI" -Device "ManipulatorIO"\
      -DeviceMap "5"

      -Name "hall_sensor_joint_6" -SignalType "DI" -Device "ManipulatorIO"\
      -DeviceMap "6"

      -Name "hall_sensor_joint_7" -SignalType "DI" -Device "ManipulatorIO"\
      -DeviceMap "2"

      -Name "hall_sensor_24V" -SignalType "DO" -Device "ManipulatorIO"\
      -DeviceMap "1"

      -Name "hand_CmdGripper" -SignalType "GO" -Device "Hand"\
      -Label "Hand Command Right" -DeviceMap "0-4" -Category "HandRight"\
      -Access "All" -SafeLevel "SGcmdSafeLevel"

      -Name "hand_CmdClearErr" -SignalType "DO" -Device "Hand"\
      -Label "Clear Error Right" -DeviceMap "7" -Category "HandRight"\
      -Access "All"

      -Name "hand_MaxPosition" -SignalType "GO" -Device "Hand"\
      -Label "Max Position Right" -DeviceMap "8-15" -Category "HandRight"\
      -Access "All" -Default 100

      -Name "hand_MinPosition" -SignalType "GO" -Device "Hand"\
      -Label "Min Position Right" -DeviceMap "16-23" -Category "HandRight"\
      -Access "All" -Default 50

      -Name "hand_MaxSpeed" -SignalType "GO" -Device "Hand"\
      -Label "Max Speed Right" -DeviceMap "24-31" -Category "HandRight"\
      -Access "All" -Default 200

      -Name "hand_HoldForce" -SignalType "GO" -Device "Hand"\
      -Label "Hold Force Right" -DeviceMap "40-47" -Category "HandRight"\
      -Access "All" -Default 120

      -Name "hand_CmdVacuum1" -SignalType "DO" -Device "Hand"\
      -Label "Vacuum 1 Right" -DeviceMap "48" -Category "HandRight"\
      -Access "All"

      -Name "hand_CmdVacuum2" -SignalType "DO" -Device "Hand"\
      -Label "Vacuum 2 Right" -DeviceMap "49" -Category "HandRight"\
      -Access "All"

      -Name "hand_CmdBlowoff1" -SignalType "DO" -Device "Hand"\
      -Label "BlowOff 1 Right" -DeviceMap "50" -Category "HandRight"\
      -Access "All"

      -Name "hand_CmdBlowoff2" -SignalType "DO" -Device "Hand"\
      -Label "BlowOff 2 Right" -DeviceMap "51" -Category "HandRight"\
      -Access "All"

      -Name "hand_simWaitState" -SignalType "DO" -Device "Hand"\
      -Label "Sim Waitstate Right" -DeviceMap "52" -Category "HandRight"\
      -Access "All"

      -Name "di_VirtuallyConnected" -SignalType "DI" -Device "Hand"\
      -Label "Virtual Controller" -DeviceMap "6" -Category "HandRight"\
      -Access "All"

      -Name "hand_SysState" -SignalType "GI" -Device "Hand"\
      -Label "Finger State Right" -DeviceMap "0-4" -Category "HandRight"\
      -Access "All"

      -Name "hand_SysError" -SignalType "GI" -Device "Hand"\
      -Label "Finger Error Right" -DeviceMap "32-39" -Category "HandRight"\
      -Access "All"

      -Name "hand_StatusCalibrated" -SignalType "DI" -Device "Hand"\
      -Label "Calibrated Right" -DeviceMap "5" -Category "HandRight"\
      -Access "All"

      -Name "hand_ActualPosition" -SignalType "GI" -Device "Hand"\
      -Label "Actual Position Right" -DeviceMap "8-15" -Category "HandRight"\
      -Access "All"

      -Name "hand_ActualSpeed" -SignalType "GI" -Device "Hand"\
      -Label "Actual Speed Right" -DeviceMap "16-23" -Category "HandRight"\
      -Access "All"

      -Name "hand_StatusCamLinked" -SignalType "DI" -Device "Hand"\
      -Label "Camera Connection Right" -DeviceMap "40" -Category "HandRight"\
      -Access "All"

      -Name "hand_SoftwareVersion" -SignalType "GI" -Device "Hand"\
      -Label "Software Version Right" -DeviceMap "41-47" -Category "HandRight"\
      -Access "All"

      -Name "hand_StatusVacuum1" -SignalType "DI" -Device "Hand"\
      -Label "Vacuum 1 Right Status" -DeviceMap "48" -Category "HandRight"\
      -Access "All"

      -Name "hand_StatusVacuum2" -SignalType "DI" -Device "Hand"\
      -Label "Vacuum 1 Right Status" -DeviceMap "49" -Category "HandRight"\
      -Access "All"

      -Name "hand_StatusBlowoff1" -SignalType "DI" -Device "Hand"\
      -Label "SuncTool 1 Right Status" -DeviceMap "50" -Category "HandRight"\
      -Access "All"

      -Name "hand_StatusBlowoff2" -SignalType "DI" -Device "Hand"\
      -Label "SuncTool 1 Right Status" -DeviceMap "51" -Category "HandRight"\
      -Access "All"

      -Name "hand_ActualPressure1" -SignalType "GI" -Device "Hand"\
      -Label "Vacuum pressure1 Right" -DeviceMap "64-71" -Category "HandRight"\
      -Access "All"

      -Name "hand_ActualPressure2" -SignalType "GI" -Device "Hand"\
      -Label "Vacuum pressure2 Right" -DeviceMap "72-79" -Category "HandRight"\
      -Access "All"

      -Name "hand_SecurityKey" -SignalType "GO" -Device "Hand"\
      -Label "Security key right" -DeviceMap "64-71" -Category "HandRight"\
      -Access "All"

      -Name "hand_TftPFtpMode" -SignalType "DI" -Device "Hand"\
      -Label "Hand firmware update mode" -DeviceMap "7" -Category "HandRight"\
      -Access "All"

      -Name "CabinetIO_0_DO1" -SignalType "DO" -Device "CabinetIO"\
      -DeviceMap "0" -Access "All"

      -Name "CabinetIO_0_DO2" -SignalType "DO" -Device "CabinetIO"\
      -DeviceMap "1" -Access "All"

      -Name "CabinetIO_0_DO3" -SignalType "DO" -Device "CabinetIO"\
      -DeviceMap "2" -Access "All"

      -Name "CabinetIO_0_DO4_JB01_LampBlu" -SignalType "DO" -Device "CabinetIO"\
      -Label "Lampe bleue - Boite de jonction" -DeviceMap "3" -Access "All"

      -Name "CabinetIO_0_DO5_JB01_LampOr" -SignalType "DO" -Device "CabinetIO"\
      -Label "Lampe orange - Boite de jonction" -DeviceMap "4" -Access "All"

      -Name "CabinetIO_0_DO6" -SignalType "DO" -Device "CabinetIO"\
      -DeviceMap "5" -Access "All"

      -Name "CabinetIO_0_DO7" -SignalType "DO" -Device "CabinetIO"\
      -DeviceMap "6" -Access "All"

      -Name "CabinetIO_0_DO8" -SignalType "DO" -Device "CabinetIO"\
      -DeviceMap "7" -Access "All"

      -Name "CabinetIO_0_DO9_FV0101" -SignalType "DO" -Device "CabinetIO"\
      -Label "GLI-Vérin Sorti" -DeviceMap "8" -Access "All"

      -Name "CabinetIO_0_DO10" -SignalType "DO" -Device "CabinetIO"\
      -DeviceMap "9" -Access "All"

      -Name "CabinetIO_0_DO11" -SignalType "DO" -Device "CabinetIO"\
      -DeviceMap "10" -Access "All"

      -Name "CabinetIO_0_DO12" -SignalType "DO" -Device "CabinetIO"\
      -DeviceMap "11" -Access "All"

      -Name "CabinetIO_0_DO13" -SignalType "DO" -Device "CabinetIO"\
      -DeviceMap "12" -Access "All"

      -Name "CabinetIO_0_DO14" -SignalType "DO" -Device "CabinetIO"\
      -DeviceMap "13" -Access "All"

      -Name "CabinetIO_0_DO15" -SignalType "DO" -Device "CabinetIO"\
      -DeviceMap "14" -Access "All"

      -Name "CabinetIO_0_DO16" -SignalType "DO" -Device "CabinetIO"\
      -DeviceMap "15" -Access "All"

      -Name "CabinetIO_0_DI1" -SignalType "DI" -Device "CabinetIO"\
      -DeviceMap "0" -Access "All"

      -Name "CabinetIO_0_DI2" -SignalType "DI" -Device "CabinetIO"\
      -DeviceMap "1" -Access "All"

      -Name "CabinetIO_0_DI3" -SignalType "DI" -Device "CabinetIO"\
      -DeviceMap "2" -Access "All"

      -Name "CabinetIO_0_DI4" -SignalType "DI" -Device "CabinetIO"\
      -DeviceMap "3" -Access "All"

      -Name "CabinetIO_0_DI5" -SignalType "DI" -Device "CabinetIO"\
      -DeviceMap "4" -Access "All"

      -Name "CabinetIO_0_DI6" -SignalType "DI" -Device "CabinetIO"\
      -DeviceMap "5" -Access "All"

      -Name "CabinetIO_0_DI7" -SignalType "DI" -Device "CabinetIO"\
      -DeviceMap "6" -Access "All"

      -Name "CabinetIO_0_DI8" -SignalType "DI" -Device "CabinetIO"\
      -DeviceMap "7" -Access "All"

      -Name "CabinetIO_0_DI9_ZS0101" -SignalType "DI" -Device "CabinetIO"\
      -Label "GLI-Bloc present au poussoir" -DeviceMap "8" -Access "All"

      -Name "CabinetIO_0_DI10_ZS0102" -SignalType "DI" -Device "CabinetIO"\
      -Label "GLI-Bloc oriente" -DeviceMap "9" -Access "All"

      -Name "CabinetIO_0_DI11_LSL0101" -SignalType "DI" -Device "CabinetIO"\
      -Label "GLI-Bloc present bas niveau" -DeviceMap "10" -Access "All"

      -Name "CabinetIO_0_DI12_LSH0101" -SignalType "DI" -Device "CabinetIO"\
      -Label "GLI-Bloc present haut niveau" -DeviceMap "11" -Access "All"

      -Name "CabinetIO_0_DI13_ZS0103" -SignalType "DI" -Device "CabinetIO"\
      -Label "GLI-Verin position retractee" -DeviceMap "12" -Access "All"

      -Name "CabinetIO_0_DI14_ZS0104" -SignalType "DI" -Device "CabinetIO"\
      -Label "GLI-Verin position etendue" -DeviceMap "13" -Access "All"

      -Name "CabinetIO_0_DI15" -SignalType "DI" -Device "CabinetIO"\
      -DeviceMap "14" -Access "All"

      -Name "CabinetIO_0_DI16" -SignalType "DI" -Device "CabinetIO"\
      -DeviceMap "15" -Access "All"

#CTRL_SIGNATURE:qyF0TOtvZGv8hXtX6Bo3tLi7I/OCuTXgI6c+v1qP5HZlgrVarUXdYjCyT7XoCiybDVlpc75NniWHurjgwzR2dw==

--- Backups/IRB14050/SYSPAR/PROC.cfg ---
PROC:CFG_1.0:7:0::

#CTRL_SIGNATURE:I+y2QaV15gWtHGM+5Z4idi3NiusZu29hLyokxM3ohwogLM8MfydOTWOtI2G6szFitByh5svEYsXD7agPogo+dQ==
